Universal Robots PolyScope program: HeatPTemBplus.urp

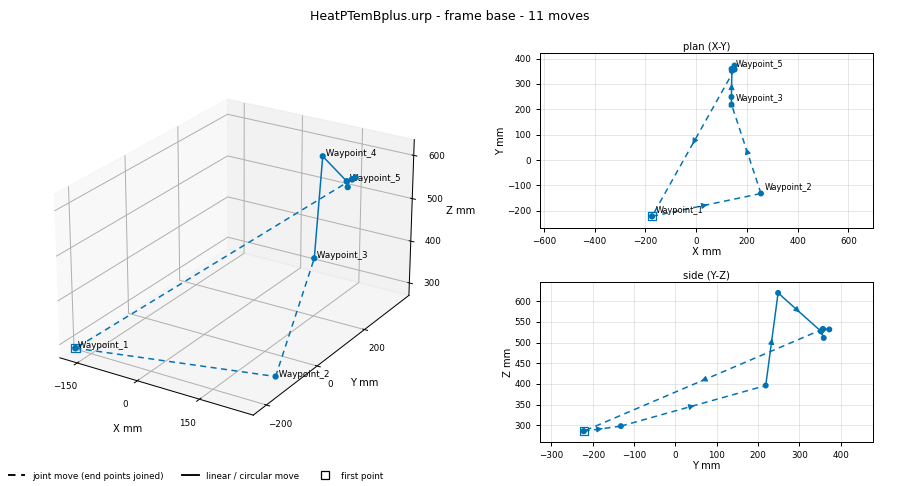
[picture p0: tool path of HeatPTemBplus.urp in frame base, 11 of 11 moves have a stored position in this frame; points joined in program order, loops and branches not executed]
Program TDHeatPTemBplus1 (installation=default directory=/programs/usbdisk_0/UR_URPs createdIn=5.11.0.108249 lastSavedIn=5.11.0.108249 robotSerialNumber=20215590035)
Calibrated DH parameters: a=[0.00016, -0.349388, -0.392209, -0.000059, 0.000026, 0]; d=[0.162575, -215.770964, 216.209801, -0.305241, 0.099656, 0.099253]; alpha=[1.570834, -0.001122, 0.007322, 1.56929, -1.570073, 0]; deltaTheta=[0, 0.606034, 5.685341, -0.008192, 0.000001, 0]
Robot Program (runOnlyOnce=true)
  MoveJ speed 60 deg/s, acceleration 80 deg/s^2 (useActiveTCP=true) feature=Base
    Waypoint Waypoint_1: TCP in base x=-173.939 y=-221.905 z=285.6 mm, rx=-2.1904 ry=-2.2352 rz=0.015 rad; joints [-99.419, -57.385, -139.029, -73.574, 89.583, 79.477] deg; TCP offset x=0 y=0 z=26 mm, rx=0 ry=0 rz=0 rad
  MoveJ speed 60 deg/s, acceleration 80 deg/s^2 (useActiveTCP=true) feature=Base
    Waypoint Waypoint_2: TCP in base x=255.607 y=-131.807 z=297.919 mm, rx=-0.0229 ry=3.1151 rz=-0.0378 rad; joints [1.04, -57.382, -137.549, -73.627, 89.053, 90.235] deg
  MoveJ speed 60 deg/s, acceleration 80 deg/s^2 (useActiveTCP=true) feature=Base
    Waypoint Waypoint_3: TCP in base x=139.565 y=218.746 z=396.126 mm, rx=-2.1977 ry=2.2399 rz=-0.0498 rad; joints [89.241, -50.957, -124.715, -95.52, 89.056, 90.235] deg
  URCap Gripper Activate (Robotiq_Grippers, Robotiq Inc.) dataModel(ResetAndActivateKey=false)
  URCap Gripper (Robotiq_Grippers, Robotiq Inc.) dataModel(position=0.0, force=99.6078431372549, speed=99.6078431372549, positionInDouble=0.0, forceInDouble=99.6078431372549, speedInDouble=99.6078431372549, slaveIds=[9], blocking=true)
  MoveP speed 250 mm/s, acceleration 1200 mm/s^2 (blendRadius=0.025 useActiveTCP=true) feature=Base
    Waypoint Waypoint_4: TCP in base x=139.138 y=248.674 z=620.253 mm, rx=-1.1946 ry=1.2372 rz=1.1708 rad; joints [89.231, -50.956, -124.823, -5.23, 88.598, 90.231] deg
  MoveL speed 250 mm/s, acceleration 1200 mm/s^2 (useActiveTCP=true) feature=Base
    Waypoint Waypoint_5: TCP in base x=140.819 y=352.481 z=527.453 mm, rx=-1.3191 ry=1.3425 rz=1.0427 rad; joints [89.895, -66.698, -128.274, 4.224, 86.527, 88.461] deg
  MoveL speed 250 mm/s, acceleration 1200 mm/s^2 (useActiveTCP=true) feature=Base
    Waypoint Waypoint_6: TCP in base x=139.623 y=359.181 z=511.306 mm, rx=-1.2848 ry=1.3105 rz=1.0646 rad; joints [90.254, -69.418, -130.155, 11.447, 86.004, 88.397] deg
  MoveL speed 250 mm/s, acceleration 1200 mm/s^2 (useActiveTCP=true) feature=Base
    Waypoint Waypoint_5: TCP in base x=140.819 y=352.481 z=527.453 mm, rx=-1.3191 ry=1.3425 rz=1.0427 rad; joints [89.895, -66.698, -128.274, 4.224, 86.527, 88.461] deg
  MoveL speed 250 mm/s, acceleration 1200 mm/s^2 (useActiveTCP=true) feature=Base
    Waypoint Waypoint_7: TCP in base x=151.132 y=357.26 z=532.747 mm, rx=-1.2834 ry=1.3929 rz=0.9577 rad; joints [89.873, -66.887, -126.734, 1.057, 81.871, 88.448] deg
  MoveL speed 250 mm/s, acceleration 1200 mm/s^2 (useActiveTCP=true) feature=Base
    Waypoint Waypoint_8: TCP in base x=151.122 y=372.678 z=531.939 mm, rx=-1.2957 ry=1.4033 rz=0.9484 rad; joints [89.873, -69.129, -125.196, 0.826, 81.885, 88.449] deg
  MoveL speed 250 mm/s, acceleration 1200 mm/s^2 (useActiveTCP=true) feature=Base
    Waypoint Waypoint_7: TCP in base x=151.132 y=357.26 z=532.747 mm, rx=-1.2834 ry=1.3929 rz=0.9577 rad; joints [89.873, -66.887, -126.734, 1.057, 81.871, 88.448] deg
  MoveJ speed 60 deg/s, acceleration 80 deg/s^2 (useActiveTCP=true) feature=Base
    Waypoint Waypoint_1: TCP in base x=-173.939 y=-221.905 z=285.6 mm, rx=-2.1904 ry=-2.2352 rz=0.015 rad; joints [-99.419, -57.385, -139.029, -73.574, 89.583, 79.477] deg
  URCap Gripper (Robotiq_Grippers, Robotiq Inc.) dataModel(position=100.0, force=99.6078431372549, speed=99.6078431372549, positionInDouble=100.0, forceInDouble=99.6078431372549, speedInDouble=99.6078431372549, slaveIds=[9], blocking=true)
